FUNCTION_BLOCK Python_Checker_Modul
VAR_IN_OUT
	
		EA_Python_Checker			: Python_Checker;
END_VAR
VAR
		
		TON_1						:TON;
		TON_2						:TON;
END_VAR



IF EA_Python_Checker.Python_Active THEN
	TON_1(IN := TRUE, PT := T#5000MS);

	IF TON_1.Q THEN
		EA_Python_Checker.Test := TRUE;
		TON_1(In := FALSE);
	END_IF

	TON_2(IN := EA_Python_Checker.Test, PT := T#5000MS);

	IF TON_2.Q THEN 
		EA_Python_Checker.Python_ERROR := TRUE;
		EA_Python_Checker.Python_Active := FALSE;
		TON_2(In := FALSE);
	END_IF
	
ELSE
	TON_1(In := FALSE);
	EA_Python_Checker.Test := FALSE; 


END_IF

END_FUNCTION_BLOCK

(* stored: Version 1.1.0.1, ProductVersion 3.1.4024.12
   POU Python_Checker_Modul: Id {0da26595-c785-4b84-9411-3e05aa8050db}, SpecialFunc None *)
